# EPICS autosave request: iocBoot/ioc13Saturn1/auto_settings.req
file "mca_settings.req",                P=$(P), M=mca1
file "dxp_settings.req",                P=$(P), R=dxp1
